// TIA Portal project "ModBus" (V17)

(* hardware
DEVICE "S7-1200 station_1"  S7-1200 Station
   slot 0: "Rack_0"  S7-1200 Rack  Rack  V1.0
   slot 1: "PLC_1"  CPU 1212C DC/DC/Rly  6ES7 212-1HE40-0XB0  V4.5
*)

// ===== PLC "PLC_1"  CPU 1212C DC/DC/Rly =====

VAR_GLOBAL   // PLC tag table "Default tag table"
   "Relay#1" AT %Q0.0 : Bool;
   "Relay#2" AT %Q0.1 : Bool;
   "Relay#3" AT %Q0.2 : Bool;
   "Relay#4" AT %Q0.3 : Bool;
   "Relay#5" AT %Q0.4 : Bool;
   "Relay#6" AT %Q0.5 : Bool;
   "Relay#7" AT %Q0.6 : Bool;
   "Relay#8" AT %Q0.7 : Bool;
END_VAR

DATA_BLOCK "MD_DB"   // DB1
{ S7_Optimized_Access := 'TRUE' }
VERSION : 0.1
   VAR
      HOLD_REG : Array[0..49] of Int;
      CONNECT : TCON_IP_v4;
      ERROR : Bool;
      STATUS : Word;
   END_VAR
BEGIN
   CONNECT.InterfaceId := 64;
   CONNECT.ID := 1;
   CONNECT.ConnectionType := 11;
   CONNECT.LocalPort := 502;
   CONNECT.RemotePort := 502;
END_DATA_BLOCK

ORGANIZATION_BLOCK "Main"   // OB1, LAD, ProgramCycle
TITLE = "Main Program Sweep (Cycle)"
{ S7_Optimized_Access := 'TRUE' }
VERSION : 0.1
   VAR_INPUT
      Initial_Call : Bool;   // Initial call of this OB
      Remanence : Bool;   // =True, if remanent data are available
   END_VAR
BEGIN

REGION Network 1
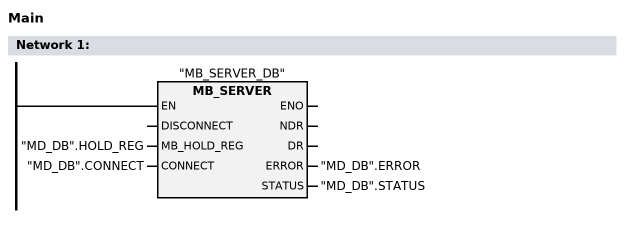
   "MB_SERVER_DB"(MB_HOLD_REG := "MD_DB".HOLD_REG,   // MB_SERVER
                  CONNECT := "MD_DB".CONNECT,
                  ERROR => "MD_DB".ERROR,
                  STATUS => "MD_DB".STATUS);
END_REGION
END_ORGANIZATION_BLOCK